{attribute 'qualified_only'}
VAR_GLOBAL CONSTANT
	IP_JANITZA: STRING(16) := '192.168.1.52';
	MBPort_Janitza : UINT := 502;
	
	b_ThirdOutputFieldAvailable	: BOOL 	:=	TRUE;
	b_InputFieldsAvailable		: BOOL	:=	TRUE;
END_VAR

(* stored: Version 1.1.0.1, ProductVersion 3.1.4024.12
   GVL PowerMeterConfig: Id {d5c3e5ba-b3df-4763-80e7-ceec20d414c0}, ParameterList True *)
